{attribute 'linkalways'} 
{attribute 'no_explicit_call' := 'This FB is a CLASS and must be accessed using methods or properties'}
{attribute 'enable_dynamic_creation'}
FUNCTION_BLOCK Node_F_VN_MedianElementElementwise_USINT EXTENDS VisionNode
VAR
    ipContainer : _ITcVnContainer;
    nMedian : _USINT(0);
    hrPrev : _HRESULT(S_OK);
    hresult : _HRESULT(S_OK);
END_VAR

METHOD PUBLIC  Clone : I_Node
VAR
	pNode : POINTER TO Node_F_VN_MedianElementElementwise_USINT;
END_VAR
pNode := __NEW(Node_F_VN_MedianElementElementwise_USINT);
Clone := pNode^;
END_METHOD

METHOD FB_init : BOOL
VAR_INPUT
	bInitRetains : BOOL; // if TRUE, the retain variables are initialized (warm start / cold start)
	bInCopyCode : BOOL;  // if TRUE, the instance afterwards gets moved into the copy code (online change)
END_VAR
AddInput('ipContainer', ipContainer);
AddInput('hrPrev', hrPrev);
AddOutput('ipContainer', ipContainer);
AddOutput('nMedian', nMedian);
AddOutput('hresult',hresult);
END_METHOD

METHOD PROTECTED OnExecute
hresult.Value := F_VN_MedianElementElementwise_USINT(
    ipContainer := ipContainer.Value,
    nMedian := nMedian.Value,
    hrPrev:= hrPrev.Value);
END_METHOD

METHOD PUBLIC PreExecutionCheck
VAR_INPUT
	Check : I_PreExecutionChecks;
END_VAR
Check.IsTrue(ipContainer.IsValid, 'ipContainer must be a valid container');
Check.IsTrue(ipContainer.IsType(TC_GLOBAL_CONST_LIST.ContainerType_Vector_USINT), 'ipContainer contains incorrect type');
END_METHOD

END_FUNCTION_BLOCK

(* stored: Version 1.1.0.1, ProductVersion 3.1.4026.13
   POU Node_F_VN_MedianElementElementwise_USINT: Id {74feff81-74da-46fb-a65e-5172a1d7e7bf}, SpecialFunc None
   Folder Constructor: Id {01c6ce87-6d33-47e8-a5c4-9f9184162ebf}
   Method Clone: Id {d077988c-efa3-4e1c-a7ab-4e671b05e764}
   Method FB_init: Id {16c62018-a913-4658-8032-afb7231f6701}
   Method OnExecute: Id {e32f94a5-2da3-4b12-a11a-7dfb5dcfd2e6}
   Method PreExecutionCheck: Id {684d313a-57cc-4476-a009-c80354a264bf} *)
